{attribute 'GeneratedUsingTerminal: EL7342-0000-0023'}
{attribute addProperty BoxType "EL7342-0000-0023"}
{attribute addProperty Id "EnableBOOL1ResetBOOL1Reduce_torqueBOOL1Threshold_activeBOOL1"}
{attribute addProperty CRC "1256562370"}
{attribute addProperty Size "4"}
TYPE Control_4AE59EC2 :
STRUCT
	{attribute addProperty Name "Enable"}
	Enable : BOOL;
	{attribute addProperty Name "Reset"}
	Reset : BOOL;
	{attribute addProperty Name "Reduce_torque"}
	Reduce_torque : BOOL;
	{attribute addProperty Name "Threshold_active"}
	Threshold_active : BOOL;
END_STRUCT
END_TYPE

(* stored: Version 1.2.0.0, ProductVersion 3.1.4024.9
   DUT Control_4AE59EC2: Id {52cd629d-5dce-4028-8c37-688269e2a3d8} *)
